# EPICS substitutions: ek9000App/Db/EL1184_mbbiDirect.substitutions
file EL1184.template
{       pattern
        {
                TERMINAL,

        }
        {
        }
}
